      FUNCTION_BLOCK FB_Scheduler_F21
      VAR_INPUT
          currH : WORD;
          currM : WORD;
          currD : WORD;
      END_VAR
      VAR_IN_OUT
          FB_Bacnet : FB_BACnet_DAIKIN_MasterStation_III_No_5;
          FB_Bacnet_b : FB_BACnet_DAIKIN_MasterStation_III_No_6;
      END_VAR
      VAR
          i : INT;
          bUnitTriggered : BOOL := FALSE; // New flag to track execution
          prevMinute : WORD := 0;        // New variable to track the previous minute
      END_VAR
      VAR PERSISTENT
          //scheduler var
          bEnSchedF21_ : BOOL := FALSE;
          wSchedWDHourStartF21_ : WORD; 
          wSchedWDMinStartF21_ : WORD; 
          wSchedWEHourStartF21_ : WORD; 
          wSchedWEMinStartF21_ : WORD;
          wSchedWDHourEndF21_ : WORD;
          wSchedWDMinEndF21_ : WORD;
          wSchedWEHourEndF21_ : WORD;
          wSchedWEMinEndF21_ : WORD;
          //unit var
          bUnitF21_ : ARRAY [1..23] OF BOOL;
      END_VAR


        // Reset trigger flag at minute change or at the exact scheduled time
        IF currM <> prevMinute OR 
           (currH = wSchedWDHourStartF21_ AND currM = wSchedWDMinStartF21_) OR 
           (currH = wSchedWDHourEndF21_ AND currM = wSchedWDMinEndF21_) THEN
            bUnitTriggered := FALSE;
            prevMinute := currM;
        END_IF

        // Unit Schedule Enable
        IF bEnSchedF21_ THEN
            // Weekday schedule
            IF currD >= 1 AND currD <= 5 THEN
                IF (wSchedWDHourStartF21_ <> wSchedWDHourEndF21_ OR wSchedWDMinStartF21_ <> wSchedWDMinEndF21_) THEN
                    // Schedule Unit ON
                    IF wSchedWDHourStartF21_ = currH AND wSchedWDMinStartF21_ = currM AND NOT bUnitTriggered THEN
                        bUnitTriggered := TRUE;
                        FOR i := 1 TO 23 DO
                            // Send command unit ON
                            IF bUnitF21_[i] THEN 
                                CASE i OF
                                    1: 
                                        
                                        FB_Bacnet.StartStopCommand_192.bEnWrite := TRUE;
                                        FB_Bacnet.StartStopCommand_192.bVal := TRUE;
                                    2: 
                                        
                                        FB_Bacnet.StartStopCommand_193.bEnWrite := TRUE;
                                        FB_Bacnet.StartStopCommand_193.bVal := TRUE;
                                    3: 
                                        
                                        FB_Bacnet.StartStopCommand_194.bEnWrite := TRUE;
                                        FB_Bacnet.StartStopCommand_194.bVal := TRUE;
                                    4: 
                                        
                                        FB_Bacnet.StartStopCommand_195.bEnWrite := TRUE;
                                        FB_Bacnet.StartStopCommand_195.bVal := TRUE;
                                    5: 
                                        
                                        FB_Bacnet.StartStopCommand_196.bEnWrite := TRUE;
                                        FB_Bacnet.StartStopCommand_196.bVal := TRUE;
                                    6: 
                                        
                                        FB_Bacnet.StartStopCommand_197.bEnWrite := TRUE;
                                        FB_Bacnet.StartStopCommand_197.bVal := TRUE;
                                    7: 
                                        
                                        FB_Bacnet.StartStopCommand_198.bEnWrite := TRUE;
                                        FB_Bacnet.StartStopCommand_198.bVal := TRUE;
                                    8: 
                                        
                                        FB_Bacnet.StartStopCommand_199.bEnWrite := TRUE;
                                        FB_Bacnet.StartStopCommand_199.bVal := TRUE;
                                    9: 
                                        
                                        FB_Bacnet.StartStopCommand_200.bEnWrite := TRUE;
                                        FB_Bacnet.StartStopCommand_200.bVal := TRUE;
                                    10: 
                                        
                                        FB_Bacnet.StartStopCommand_201.bEnWrite := TRUE;
                                        FB_Bacnet.StartStopCommand_201.bVal := TRUE;
                                    11: 
                                        
                                        FB_Bacnet.StartStopCommand_202.bEnWrite := TRUE;
                                        FB_Bacnet.StartStopCommand_202.bVal := TRUE;
                                    12: 
                                        
                                        FB_Bacnet.StartStopCommand_203.bEnWrite := TRUE;
                                        FB_Bacnet.StartStopCommand_203.bVal := TRUE;
                                    13: 
                                        
                                        FB_Bacnet.StartStopCommand_204.bEnWrite := TRUE;
                                        FB_Bacnet.StartStopCommand_204.bVal := TRUE;
                                    14: 
                                        
                                        FB_Bacnet.StartStopCommand_205.bEnWrite := TRUE;
                                        FB_Bacnet.StartStopCommand_205.bVal := TRUE;
                                    15: 
                                        
                                        FB_Bacnet.StartStopCommand_206.bEnWrite := TRUE;
                                        FB_Bacnet.StartStopCommand_206.bVal := TRUE;
                                    16: 
                                        
                                        FB_Bacnet.StartStopCommand_207.bEnWrite := TRUE;
                                        FB_Bacnet.StartStopCommand_207.bVal := TRUE;
                                    17: 
                                        
                                        FB_Bacnet.StartStopCommand_208.bEnWrite := TRUE;
                                        FB_Bacnet.StartStopCommand_208.bVal := TRUE;
                                    18: 
                                        
                                        FB_Bacnet.StartStopCommand_209.bEnWrite := TRUE;
                                        FB_Bacnet.StartStopCommand_209.bVal := TRUE;
                                    19: 
                                        
                                        FB_Bacnet.StartStopCommand_210.bEnWrite := TRUE;
                                        FB_Bacnet.StartStopCommand_210.bVal := TRUE;
                                    20: 
                                        
                                        FB_Bacnet.StartStopCommand_211.bEnWrite := TRUE;
                                        FB_Bacnet.StartStopCommand_211.bVal := TRUE;
                                    21: 
                                        
                                        FB_Bacnet.StartStopCommand_240.bEnWrite := TRUE;
                                        FB_Bacnet.StartStopCommand_240.bVal := TRUE;
                                    22: 
                                        
                                        FB_Bacnet_b.StartStopCommand_049.bEnWrite := TRUE;
                                        FB_Bacnet_b.StartStopCommand_049.bVal := TRUE;
                                    23: 
                                        
                                        FB_Bacnet_b.StartStopCommand_034.bEnWrite := TRUE;
                                        FB_Bacnet_b.StartStopCommand_034.bVal := TRUE;
                                END_CASE
                            END_IF
                        END_FOR
                    END_IF
                    // Schedule Unit OFF
                    IF wSchedWDHourEndF21_ = currH AND wSchedWDMinEndF21_ = currM AND NOT bUnitTriggered THEN
                        bUnitTriggered := TRUE;
                        FOR i := 1 TO 23 DO
                            // Send command unit OFF
                            IF bUnitF21_[i] THEN 
                                CASE i OF
                                    1: 
                                        
                                        FB_Bacnet.StartStopCommand_192.bEnWrite := TRUE;
                                        FB_Bacnet.StartStopCommand_192.bVal := FALSE;
                                    2: 
                                        
                                        FB_Bacnet.StartStopCommand_193.bEnWrite := TRUE;
                                        FB_Bacnet.StartStopCommand_193.bVal := FALSE;
                                    3: 
                                        
                                        FB_Bacnet.StartStopCommand_194.bEnWrite := TRUE;
                                        FB_Bacnet.StartStopCommand_194.bVal := FALSE;
                                    4: 
                                        
                                        FB_Bacnet.StartStopCommand_195.bEnWrite := TRUE;
                                        FB_Bacnet.StartStopCommand_195.bVal := FALSE;
                                    5: 
                                        
                                        FB_Bacnet.StartStopCommand_196.bEnWrite := TRUE;
                                        FB_Bacnet.StartStopCommand_196.bVal := FALSE;
                                    6: 
                                        
                                        FB_Bacnet.StartStopCommand_197.bEnWrite := TRUE;
                                        FB_Bacnet.StartStopCommand_197.bVal := FALSE;
                                    7: 
                                        
                                        FB_Bacnet.StartStopCommand_198.bEnWrite := TRUE;
                                        FB_Bacnet.StartStopCommand_198.bVal := FALSE;
                                    8: 
                                        
                                        FB_Bacnet.StartStopCommand_199.bEnWrite := TRUE;
                                        FB_Bacnet.StartStopCommand_199.bVal := FALSE;
                                    9: 
                                        
                                        FB_Bacnet.StartStopCommand_200.bEnWrite := TRUE;
                                        FB_Bacnet.StartStopCommand_200.bVal := FALSE;
                                    10: 
                                        
                                        FB_Bacnet.StartStopCommand_201.bEnWrite := TRUE;
                                        FB_Bacnet.StartStopCommand_201.bVal := FALSE;
                                    11: 
                                        
                                        FB_Bacnet.StartStopCommand_202.bEnWrite := TRUE;
                                        FB_Bacnet.StartStopCommand_202.bVal := FALSE;
                                    12: 
                                        
                                        FB_Bacnet.StartStopCommand_203.bEnWrite := TRUE;
                                        FB_Bacnet.StartStopCommand_203.bVal := FALSE;
                                    13: 
                                        
                                        FB_Bacnet.StartStopCommand_204.bEnWrite := TRUE;
                                        FB_Bacnet.StartStopCommand_204.bVal := FALSE;
                                    14: 
                                        
                                        FB_Bacnet.StartStopCommand_205.bEnWrite := TRUE;
                                        FB_Bacnet.StartStopCommand_205.bVal := FALSE;
                                    15: 
                                        
                                        FB_Bacnet.StartStopCommand_206.bEnWrite := TRUE;
                                        FB_Bacnet.StartStopCommand_206.bVal := FALSE;
                                    16: 
                                        
                                        FB_Bacnet.StartStopCommand_207.bEnWrite := TRUE;
                                        FB_Bacnet.StartStopCommand_207.bVal := FALSE;
                                    17: 
                                        
                                        FB_Bacnet.StartStopCommand_208.bEnWrite := TRUE;
                                        FB_Bacnet.StartStopCommand_208.bVal := FALSE;
                                    18: 
                                        
                                        FB_Bacnet.StartStopCommand_209.bEnWrite := TRUE;
                                        FB_Bacnet.StartStopCommand_209.bVal := FALSE;
                                    19: 
                                        
                                        FB_Bacnet.StartStopCommand_210.bEnWrite := TRUE;
                                        FB_Bacnet.StartStopCommand_210.bVal := FALSE;
                                    20: 
                                        
                                        FB_Bacnet.StartStopCommand_211.bEnWrite := TRUE;
                                        FB_Bacnet.StartStopCommand_211.bVal := FALSE;
                                    21: 
                                        
                                        FB_Bacnet.StartStopCommand_240.bEnWrite := TRUE;
                                        FB_Bacnet.StartStopCommand_240.bVal := FALSE;
                                    22: 
                                        
                                        FB_Bacnet_b.StartStopCommand_049.bEnWrite := TRUE;
                                        FB_Bacnet_b.StartStopCommand_049.bVal := FALSE;
                                    23: 
                                        
                                        FB_Bacnet_b.StartStopCommand_034.bEnWrite := TRUE;
                                        FB_Bacnet_b.StartStopCommand_034.bVal := FALSE;
                                END_CASE
                            END_IF
                        END_FOR
                    END_IF
                END_IF
            END_IF

            // Weekend schedule
            IF currD = 0 OR currD = 6 THEN
                IF (wSchedWEHourStartF21_ <> wSchedWEHourEndF21_ OR wSchedWEMinStartF21_ <> wSchedWEMinEndF21_) THEN
                    // Schedule Unit ON
                    IF wSchedWEHourStartF21_ = currH AND wSchedWEMinStartF21_ = currM AND NOT bUnitTriggered THEN
                        bUnitTriggered := TRUE;
                        FOR i := 1 TO 23 DO
                            // Send command unit ON
                            IF bUnitF21_[i] THEN 
                                CASE i OF
                                    1: 
                                        
                                        FB_Bacnet.StartStopCommand_192.bEnWrite := TRUE;
                                        FB_Bacnet.StartStopCommand_192.bVal := TRUE;
                                    2: 
                                        
                                        FB_Bacnet.StartStopCommand_193.bEnWrite := TRUE;
                                        FB_Bacnet.StartStopCommand_193.bVal := TRUE;
                                    3: 
                                        
                                        FB_Bacnet.StartStopCommand_194.bEnWrite := TRUE;
                                        FB_Bacnet.StartStopCommand_194.bVal := TRUE;
                                    4: 
                                        
                                        FB_Bacnet.StartStopCommand_195.bEnWrite := TRUE;
                                        FB_Bacnet.StartStopCommand_195.bVal := TRUE;
                                    5: 
                                        
                                        FB_Bacnet.StartStopCommand_196.bEnWrite := TRUE;
                                        FB_Bacnet.StartStopCommand_196.bVal := TRUE;
                                    6: 
                                        
                                        FB_Bacnet.StartStopCommand_197.bEnWrite := TRUE;
                                        FB_Bacnet.StartStopCommand_197.bVal := TRUE;
                                    7: 
                                        
                                        FB_Bacnet.StartStopCommand_198.bEnWrite := TRUE;
                                        FB_Bacnet.StartStopCommand_198.bVal := TRUE;
                                    8: 
                                        
                                        FB_Bacnet.StartStopCommand_199.bEnWrite := TRUE;
                                        FB_Bacnet.StartStopCommand_199.bVal := TRUE;
                                    9: 
                                        
                                        FB_Bacnet.StartStopCommand_200.bEnWrite := TRUE;
                                        FB_Bacnet.StartStopCommand_200.bVal := TRUE;
                                    10: 
                                        
                                        FB_Bacnet.StartStopCommand_201.bEnWrite := TRUE;
                                        FB_Bacnet.StartStopCommand_201.bVal := TRUE;
                                    11: 
                                        
                                        FB_Bacnet.StartStopCommand_202.bEnWrite := TRUE;
                                        FB_Bacnet.StartStopCommand_202.bVal := TRUE;
                                    12: 
                                        
                                        FB_Bacnet.StartStopCommand_203.bEnWrite := TRUE;
                                        FB_Bacnet.StartStopCommand_203.bVal := TRUE;
                                    13: 
                                        
                                        FB_Bacnet.StartStopCommand_204.bEnWrite := TRUE;
                                        FB_Bacnet.StartStopCommand_204.bVal := TRUE;
                                    14: 
                                        
                                        FB_Bacnet.StartStopCommand_205.bEnWrite := TRUE;
                                        FB_Bacnet.StartStopCommand_205.bVal := TRUE;
                                    15: 
                                        
                                        FB_Bacnet.StartStopCommand_206.bEnWrite := TRUE;
                                        FB_Bacnet.StartStopCommand_206.bVal := TRUE;
                                    16: 
                                        
                                        FB_Bacnet.StartStopCommand_207.bEnWrite := TRUE;
                                        FB_Bacnet.StartStopCommand_207.bVal := TRUE;
                                    17: 
                                        
                                        FB_Bacnet.StartStopCommand_208.bEnWrite := TRUE;
                                        FB_Bacnet.StartStopCommand_208.bVal := TRUE;
                                    18: 
                                        
                                        FB_Bacnet.StartStopCommand_209.bEnWrite := TRUE;
                                        FB_Bacnet.StartStopCommand_209.bVal := TRUE;
                                    19: 
                                        
                                        FB_Bacnet.StartStopCommand_210.bEnWrite := TRUE;
                                        FB_Bacnet.StartStopCommand_210.bVal := TRUE;
                                    20: 
                                        
                                        FB_Bacnet.StartStopCommand_211.bEnWrite := TRUE;
                                        FB_Bacnet.StartStopCommand_211.bVal := TRUE;
                                    21: 
                                        
                                        FB_Bacnet.StartStopCommand_240.bEnWrite := TRUE;
                                        FB_Bacnet.StartStopCommand_240.bVal := TRUE;
                                    22: 
                                        
                                        FB_Bacnet_b.StartStopCommand_049.bEnWrite := TRUE;
                                        FB_Bacnet_b.StartStopCommand_049.bVal := TRUE;
                                    23: 
                                        
                                        FB_Bacnet_b.StartStopCommand_034.bEnWrite := TRUE;
                                        FB_Bacnet_b.StartStopCommand_034.bVal := TRUE;
                                END_CASE
                            END_IF
                        END_FOR
                    END_IF
                    // Schedule Unit OFF
                    IF wSchedWEHourEndF21_ = currH AND wSchedWEMinEndF21_ = currM AND NOT bUnitTriggered THEN
                        bUnitTriggered := TRUE;
                        FOR i := 1 TO 23 DO
                            // Send command unit OFF
                            IF bUnitF21_[i] THEN 
                                CASE i OF
                                    1: 
                                        
                                        FB_Bacnet.StartStopCommand_192.bEnWrite := TRUE;
                                        FB_Bacnet.StartStopCommand_192.bVal := FALSE;
                                    2: 
                                        
                                        FB_Bacnet.StartStopCommand_193.bEnWrite := TRUE;
                                        FB_Bacnet.StartStopCommand_193.bVal := FALSE;
                                    3: 
                                        
                                        FB_Bacnet.StartStopCommand_194.bEnWrite := TRUE;
                                        FB_Bacnet.StartStopCommand_194.bVal := FALSE;
                                    4: 
                                        
                                        FB_Bacnet.StartStopCommand_195.bEnWrite := TRUE;
                                        FB_Bacnet.StartStopCommand_195.bVal := FALSE;
                                    5: 
                                        
                                        FB_Bacnet.StartStopCommand_196.bEnWrite := TRUE;
                                        FB_Bacnet.StartStopCommand_196.bVal := FALSE;
                                    6: 
                                        
                                        FB_Bacnet.StartStopCommand_197.bEnWrite := TRUE;
                                        FB_Bacnet.StartStopCommand_197.bVal := FALSE;
                                    7: 
                                        
                                        FB_Bacnet.StartStopCommand_198.bEnWrite := TRUE;
                                        FB_Bacnet.StartStopCommand_198.bVal := FALSE;
                                    8: 
                                        
                                        FB_Bacnet.StartStopCommand_199.bEnWrite := TRUE;
                                        FB_Bacnet.StartStopCommand_199.bVal := FALSE;
                                    9: 
                                        
                                        FB_Bacnet.StartStopCommand_200.bEnWrite := TRUE;
                                        FB_Bacnet.StartStopCommand_200.bVal := FALSE;
                                    10: 
                                        
                                        FB_Bacnet.StartStopCommand_201.bEnWrite := TRUE;
                                        FB_Bacnet.StartStopCommand_201.bVal := FALSE;
                                    11: 
                                        
                                        FB_Bacnet.StartStopCommand_202.bEnWrite := TRUE;
                                        FB_Bacnet.StartStopCommand_202.bVal := FALSE;
                                    12: 
                                        
                                        FB_Bacnet.StartStopCommand_203.bEnWrite := TRUE;
                                        FB_Bacnet.StartStopCommand_203.bVal := FALSE;
                                    13: 
                                        
                                        FB_Bacnet.StartStopCommand_204.bEnWrite := TRUE;
                                        FB_Bacnet.StartStopCommand_204.bVal := FALSE;
                                    14: 
                                        
                                        FB_Bacnet.StartStopCommand_205.bEnWrite := TRUE;
                                        FB_Bacnet.StartStopCommand_205.bVal := FALSE;
                                    15: 
                                        
                                        FB_Bacnet.StartStopCommand_206.bEnWrite := TRUE;
                                        FB_Bacnet.StartStopCommand_206.bVal := FALSE;
                                    16: 
                                        
                                        FB_Bacnet.StartStopCommand_207.bEnWrite := TRUE;
                                        FB_Bacnet.StartStopCommand_207.bVal := FALSE;
                                    17: 
                                        
                                        FB_Bacnet.StartStopCommand_208.bEnWrite := TRUE;
                                        FB_Bacnet.StartStopCommand_208.bVal := FALSE;
                                    18: 
                                        
                                        FB_Bacnet.StartStopCommand_209.bEnWrite := TRUE;
                                        FB_Bacnet.StartStopCommand_209.bVal := FALSE;
                                    19: 
                                        
                                        FB_Bacnet.StartStopCommand_210.bEnWrite := TRUE;
                                        FB_Bacnet.StartStopCommand_210.bVal := FALSE;
                                    20: 
                                        
                                        FB_Bacnet.StartStopCommand_211.bEnWrite := TRUE;
                                        FB_Bacnet.StartStopCommand_211.bVal := FALSE;
                                    21: 
                                        
                                        FB_Bacnet.StartStopCommand_240.bEnWrite := TRUE;
                                        FB_Bacnet.StartStopCommand_240.bVal := FALSE;
                                    22: 
                                        
                                        FB_Bacnet_b.StartStopCommand_049.bEnWrite := TRUE;
                                        FB_Bacnet_b.StartStopCommand_049.bVal := FALSE;
                                    23: 
                                        
                                        FB_Bacnet_b.StartStopCommand_034.bEnWrite := TRUE;
                                        FB_Bacnet_b.StartStopCommand_034.bVal := FALSE;
                                END_CASE
                            END_IF
                        END_FOR
                    END_IF
                END_IF
            END_IF
        END_IF

END_FUNCTION_BLOCK

// ---- POUs/FB_Scheduler/FB_Scheduler_F22.TcPOU

      FUNCTION_BLOCK FB_Scheduler_F22
      VAR_INPUT
          currH : WORD;
          currM : WORD;
          currD : WORD;
      END_VAR
      VAR_IN_OUT
          FB_Bacnet : FB_BACnet_DAIKIN_MasterStation_III_No_6;
      END_VAR
      VAR
          i : INT;
          bUnitTriggered : BOOL := FALSE; // New flag to track execution
          prevMinute : WORD := 0;        // New variable to track the previous minute
      END_VAR
      VAR PERSISTENT
          //scheduler var
          bEnSchedF22_ : BOOL := FALSE;
          wSchedWDHourStartF22_ : WORD; 
          wSchedWDMinStartF22_ : WORD; 
          wSchedWEHourStartF22_ : WORD; 
          wSchedWEMinStartF22_ : WORD;
          wSchedWDHourEndF22_ : WORD;
          wSchedWDMinEndF22_ : WORD;
          wSchedWEHourEndF22_ : WORD;
          wSchedWEMinEndF22_ : WORD;
          //unit var
          bUnitF22_ : ARRAY [1..21] OF BOOL;
      END_VAR


        // Reset trigger flag at minute change or at the exact scheduled time
        IF currM <> prevMinute OR 
           (currH = wSchedWDHourStartF22_ AND currM = wSchedWDMinStartF22_) OR 
           (currH = wSchedWDHourEndF22_ AND currM = wSchedWDMinEndF22_) THEN
            bUnitTriggered := FALSE;
            prevMinute := currM;
        END_IF

        // Unit Schedule Enable
        IF bEnSchedF22_ THEN
            // Weekday schedule
            IF currD >= 1 AND currD <= 5 THEN
                IF (wSchedWDHourStartF22_ <> wSchedWDHourEndF22_ OR wSchedWDMinStartF22_ <> wSchedWDMinEndF22_) THEN
                    // Schedule Unit ON
                    IF wSchedWDHourStartF22_ = currH AND wSchedWDMinStartF22_ = currM AND NOT bUnitTriggered THEN
                        bUnitTriggered := TRUE;
                        FOR i := 1 TO 21 DO
                            // Send command unit ON
                            IF bUnitF22_[i] THEN 
                                CASE i OF
                                    1: 
                                        
                                        FB_Bacnet.StartStopCommand_000.bEnWrite := TRUE;
                                        FB_Bacnet.StartStopCommand_000.bVal := TRUE;
                                    2: 
                                        
                                        FB_Bacnet.StartStopCommand_001.bEnWrite := TRUE;
                                        FB_Bacnet.StartStopCommand_001.bVal := TRUE;
                                    3: 
                                        
                                        FB_Bacnet.StartStopCommand_002.bEnWrite := TRUE;
                                        FB_Bacnet.StartStopCommand_002.bVal := TRUE;
                                    4: 
                                        
                                        FB_Bacnet.StartStopCommand_003.bEnWrite := TRUE;
                                        FB_Bacnet.StartStopCommand_003.bVal := TRUE;
                                    5: 
                                        
                                        FB_Bacnet.StartStopCommand_004.bEnWrite := TRUE;
                                        FB_Bacnet.StartStopCommand_004.bVal := TRUE;
                                    6: 
                                        
                                        FB_Bacnet.StartStopCommand_005.bEnWrite := TRUE;
                                        FB_Bacnet.StartStopCommand_005.bVal := TRUE;
                                    7: 
                                        
                                        FB_Bacnet.StartStopCommand_006.bEnWrite := TRUE;
                                        FB_Bacnet.StartStopCommand_006.bVal := TRUE;
                                    8: 
                                        
                                        FB_Bacnet.StartStopCommand_007.bEnWrite := TRUE;
                                        FB_Bacnet.StartStopCommand_007.bVal := TRUE;
                                    9: 
                                        
                                        FB_Bacnet.StartStopCommand_008.bEnWrite := TRUE;
                                        FB_Bacnet.StartStopCommand_008.bVal := TRUE;
                                    10: 
                                        
                                        FB_Bacnet.StartStopCommand_009.bEnWrite := TRUE;
                                        FB_Bacnet.StartStopCommand_009.bVal := TRUE;
                                    11: 
                                        
                                        FB_Bacnet.StartStopCommand_010.bEnWrite := TRUE;
                                        FB_Bacnet.StartStopCommand_010.bVal := TRUE;
                                    12: 
                                        
                                        FB_Bacnet.StartStopCommand_011.bEnWrite := TRUE;
                                        FB_Bacnet.StartStopCommand_011.bVal := TRUE;
                                    13: 
                                        
                                        FB_Bacnet.StartStopCommand_012.bEnWrite := TRUE;
                                        FB_Bacnet.StartStopCommand_012.bVal := TRUE;
                                    14: 
                                        
                                        FB_Bacnet.StartStopCommand_013.bEnWrite := TRUE;
                                        FB_Bacnet.StartStopCommand_013.bVal := TRUE;
                                    15: 
                                        
                                        FB_Bacnet.StartStopCommand_014.bEnWrite := TRUE;
                                        FB_Bacnet.StartStopCommand_014.bVal := TRUE;
                                    16: 
                                        
                                        FB_Bacnet.StartStopCommand_015.bEnWrite := TRUE;
                                        FB_Bacnet.StartStopCommand_015.bVal := TRUE;
                                    17: 
                                        
                                        FB_Bacnet.StartStopCommand_016.bEnWrite := TRUE;
                                        FB_Bacnet.StartStopCommand_016.bVal := TRUE;
                                    18: 
                                        
                                        FB_Bacnet.StartStopCommand_017.bEnWrite := TRUE;
                                        FB_Bacnet.StartStopCommand_017.bVal := TRUE;
                                    19: 
                                        
                                        FB_Bacnet.StartStopCommand_018.bEnWrite := TRUE;
                                        FB_Bacnet.StartStopCommand_018.bVal := TRUE;
                                    20: 
                                        
                                        FB_Bacnet.StartStopCommand_019.bEnWrite := TRUE;
                                        FB_Bacnet.StartStopCommand_019.bVal := TRUE;
                                    21: 
                                        
                                        FB_Bacnet.StartStopCommand_035.bEnWrite := TRUE;
                                        FB_Bacnet.StartStopCommand_035.bVal := TRUE;
                                END_CASE
                            END_IF
                        END_FOR
                    END_IF
                    // Schedule Unit OFF
                    IF wSchedWDHourEndF22_ = currH AND wSchedWDMinEndF22_ = currM AND NOT bUnitTriggered THEN
                        bUnitTriggered := TRUE;
                        FOR i := 1 TO 21 DO
                            // Send command unit OFF
                            IF bUnitF22_[i] THEN 
                                CASE i OF
                                    1: 
                                        
                                        FB_Bacnet.StartStopCommand_000.bEnWrite := TRUE;
                                        FB_Bacnet.StartStopCommand_000.bVal := FALSE;
                                    2: 
                                        
                                        FB_Bacnet.StartStopCommand_001.bEnWrite := TRUE;
                                        FB_Bacnet.StartStopCommand_001.bVal := FALSE;
                                    3: 
                                        
                                        FB_Bacnet.StartStopCommand_002.bEnWrite := TRUE;
                                        FB_Bacnet.StartStopCommand_002.bVal := FALSE;
                                    4: 
                                        
                                        FB_Bacnet.StartStopCommand_003.bEnWrite := TRUE;
                                        FB_Bacnet.StartStopCommand_003.bVal := FALSE;
                                    5: 
                                        
                                        FB_Bacnet.StartStopCommand_004.bEnWrite := TRUE;
                                        FB_Bacnet.StartStopCommand_004.bVal := FALSE;
                                    6: 
                                        
                                        FB_Bacnet.StartStopCommand_005.bEnWrite := TRUE;
                                        FB_Bacnet.StartStopCommand_005.bVal := FALSE;
                                    7: 
                                        
                                        FB_Bacnet.StartStopCommand_006.bEnWrite := TRUE;
                                        FB_Bacnet.StartStopCommand_006.bVal := FALSE;
                                    8: 
                                        
                                        FB_Bacnet.StartStopCommand_007.bEnWrite := TRUE;
                                        FB_Bacnet.StartStopCommand_007.bVal := FALSE;
                                    9: 
                                        
                                        FB_Bacnet.StartStopCommand_008.bEnWrite := TRUE;
                                        FB_Bacnet.StartStopCommand_008.bVal := FALSE;
                                    10: 
                                        
                                        FB_Bacnet.StartStopCommand_009.bEnWrite := TRUE;
                                        FB_Bacnet.StartStopCommand_009.bVal := FALSE;
                                    11: 
                                        
                                        FB_Bacnet.StartStopCommand_010.bEnWrite := TRUE;
                                        FB_Bacnet.StartStopCommand_010.bVal := FALSE;
                                    12: 
                                        
                                        FB_Bacnet.StartStopCommand_011.bEnWrite := TRUE;
                                        FB_Bacnet.StartStopCommand_011.bVal := FALSE;
                                    13: 
                                        
                                        FB_Bacnet.StartStopCommand_012.bEnWrite := TRUE;
                                        FB_Bacnet.StartStopCommand_012.bVal := FALSE;
                                    14: 
                                        
                                        FB_Bacnet.StartStopCommand_013.bEnWrite := TRUE;
                                        FB_Bacnet.StartStopCommand_013.bVal := FALSE;
                                    15: 
                                        
                                        FB_Bacnet.StartStopCommand_014.bEnWrite := TRUE;
                                        FB_Bacnet.StartStopCommand_014.bVal := FALSE;
                                    16: 
                                        
                                        FB_Bacnet.StartStopCommand_015.bEnWrite := TRUE;
                                        FB_Bacnet.StartStopCommand_015.bVal := FALSE;
                                    17: 
                                        
                                        FB_Bacnet.StartStopCommand_016.bEnWrite := TRUE;
                                        FB_Bacnet.StartStopCommand_016.bVal := FALSE;
                                    18: 
                                        
                                        FB_Bacnet.StartStopCommand_017.bEnWrite := TRUE;
                                        FB_Bacnet.StartStopCommand_017.bVal := FALSE;
                                    19: 
                                        
                                        FB_Bacnet.StartStopCommand_018.bEnWrite := TRUE;
                                        FB_Bacnet.StartStopCommand_018.bVal := FALSE;
                                    20: 
                                        
                                        FB_Bacnet.StartStopCommand_019.bEnWrite := TRUE;
                                        FB_Bacnet.StartStopCommand_019.bVal := FALSE;
                                    21: 
                                        
                                        FB_Bacnet.StartStopCommand_035.bEnWrite := TRUE;
                                        FB_Bacnet.StartStopCommand_035.bVal := FALSE;
                                END_CASE
                            END_IF
                        END_FOR
                    END_IF
                END_IF
            END_IF

            // Weekend schedule
            IF currD = 0 OR currD = 6 THEN
                IF (wSchedWEHourStartF22_ <> wSchedWEHourEndF22_ OR wSchedWEMinStartF22_ <> wSchedWEMinEndF22_) THEN
                    // Schedule Unit ON
                    IF wSchedWEHourStartF22_ = currH AND wSchedWEMinStartF22_ = currM AND NOT bUnitTriggered THEN
                        bUnitTriggered := TRUE;
                        FOR i := 1 TO 21 DO
                            // Send command unit ON
                            IF bUnitF22_[i] THEN 
                                CASE i OF
                                    1: 
                                        
                                        FB_Bacnet.StartStopCommand_000.bEnWrite := TRUE;
                                        FB_Bacnet.StartStopCommand_000.bVal := TRUE;
                                    2: 
                                        
                                        FB_Bacnet.StartStopCommand_001.bEnWrite := TRUE;
                                        FB_Bacnet.StartStopCommand_001.bVal := TRUE;
                                    3: 
                                        
                                        FB_Bacnet.StartStopCommand_002.bEnWrite := TRUE;
                                        FB_Bacnet.StartStopCommand_002.bVal := TRUE;
                                    4: 
                                        
                                        FB_Bacnet.StartStopCommand_003.bEnWrite := TRUE;
                                        FB_Bacnet.StartStopCommand_003.bVal := TRUE;
                                    5: 
                                        
                                        FB_Bacnet.StartStopCommand_004.bEnWrite := TRUE;
                                        FB_Bacnet.StartStopCommand_004.bVal := TRUE;
                                    6: 
                                        
                                        FB_Bacnet.StartStopCommand_005.bEnWrite := TRUE;
                                        FB_Bacnet.StartStopCommand_005.bVal := TRUE;
                                    7: 
                                        
                                        FB_Bacnet.StartStopCommand_006.bEnWrite := TRUE;
                                        FB_Bacnet.StartStopCommand_006.bVal := TRUE;
                                    8: 
                                        
                                        FB_Bacnet.StartStopCommand_007.bEnWrite := TRUE;
                                        FB_Bacnet.StartStopCommand_007.bVal := TRUE;
                                    9: 
                                        
                                        FB_Bacnet.StartStopCommand_008.bEnWrite := TRUE;
                                        FB_Bacnet.StartStopCommand_008.bVal := TRUE;
                                    10: 
                                        
                                        FB_Bacnet.StartStopCommand_009.bEnWrite := TRUE;
                                        FB_Bacnet.StartStopCommand_009.bVal := TRUE;
                                    11: 
                                        
                                        FB_Bacnet.StartStopCommand_010.bEnWrite := TRUE;
                                        FB_Bacnet.StartStopCommand_010.bVal := TRUE;
                                    12: 
                                        
                                        FB_Bacnet.StartStopCommand_011.bEnWrite := TRUE;
                                        FB_Bacnet.StartStopCommand_011.bVal := TRUE;
                                    13: 
                                        
                                        FB_Bacnet.StartStopCommand_012.bEnWrite := TRUE;
                                        FB_Bacnet.StartStopCommand_012.bVal := TRUE;
                                    14: 
                                        
                                        FB_Bacnet.StartStopCommand_013.bEnWrite := TRUE;
                                        FB_Bacnet.StartStopCommand_013.bVal := TRUE;
                                    15: 
                                        
                                        FB_Bacnet.StartStopCommand_014.bEnWrite := TRUE;
                                        FB_Bacnet.StartStopCommand_014.bVal := TRUE;
                                    16: 
                                        
                                        FB_Bacnet.StartStopCommand_015.bEnWrite := TRUE;
                                        FB_Bacnet.StartStopCommand_015.bVal := TRUE;
                                    17: 
                                        
                                        FB_Bacnet.StartStopCommand_016.bEnWrite := TRUE;
                                        FB_Bacnet.StartStopCommand_016.bVal := TRUE;
                                    18: 
                                        
                                        FB_Bacnet.StartStopCommand_017.bEnWrite := TRUE;
                                        FB_Bacnet.StartStopCommand_017.bVal := TRUE;
                                    19: 
                                        
                                        FB_Bacnet.StartStopCommand_018.bEnWrite := TRUE;
                                        FB_Bacnet.StartStopCommand_018.bVal := TRUE;
                                    20: 
                                        
                                        FB_Bacnet.StartStopCommand_019.bEnWrite := TRUE;
                                        FB_Bacnet.StartStopCommand_019.bVal := TRUE;
                                    21: 
                                        
                                        FB_Bacnet.StartStopCommand_035.bEnWrite := TRUE;
                                        FB_Bacnet.StartStopCommand_035.bVal := TRUE;
                                END_CASE
                            END_IF
                        END_FOR        
                    END_IF
                    // Schedule Unit OFF
                    IF wSchedWEHourEndF22_ = currH AND wSchedWEMinEndF22_ = currM AND NOT bUnitTriggered THEN
                        bUnitTriggered := TRUE;
                        FOR i := 1 TO 21 DO
                            // Send command unit OFF
                            IF bUnitF22_[i] THEN 
                                CASE i OF
                                    1: 
                                        
                                        FB_Bacnet.StartStopCommand_000.bEnWrite := TRUE;
                                        FB_Bacnet.StartStopCommand_000.bVal := FALSE;
                                    2: 
                                        
                                        FB_Bacnet.StartStopCommand_001.bEnWrite := TRUE;
                                        FB_Bacnet.StartStopCommand_001.bVal := FALSE;
                                    3: 
                                        
                                        FB_Bacnet.StartStopCommand_002.bEnWrite := TRUE;
                                        FB_Bacnet.StartStopCommand_002.bVal := FALSE;
                                    4: 
                                        
                                        FB_Bacnet.StartStopCommand_003.bEnWrite := TRUE;
                                        FB_Bacnet.StartStopCommand_003.bVal := FALSE;
                                    5: 
                                        
                                        FB_Bacnet.StartStopCommand_004.bEnWrite := TRUE;
                                        FB_Bacnet.StartStopCommand_004.bVal := FALSE;
                                    6: 
                                        
                                        FB_Bacnet.StartStopCommand_005.bEnWrite := TRUE;
                                        FB_Bacnet.StartStopCommand_005.bVal := FALSE;
                                    7: 
                                        
                                        FB_Bacnet.StartStopCommand_006.bEnWrite := TRUE;
                                        FB_Bacnet.StartStopCommand_006.bVal := FALSE;
                                    8: 
                                        
                                        FB_Bacnet.StartStopCommand_007.bEnWrite := TRUE;
                                        FB_Bacnet.StartStopCommand_007.bVal := FALSE;
                                    9: 
                                        
                                        FB_Bacnet.StartStopCommand_008.bEnWrite := TRUE;
                                        FB_Bacnet.StartStopCommand_008.bVal := FALSE;
                                    10: 
                                        
                                        FB_Bacnet.StartStopCommand_009.bEnWrite := TRUE;
                                        FB_Bacnet.StartStopCommand_009.bVal := FALSE;
                                    11: 
                                        
                                        FB_Bacnet.StartStopCommand_010.bEnWrite := TRUE;
                                        FB_Bacnet.StartStopCommand_010.bVal := FALSE;
                                    12: 
                                        
                                        FB_Bacnet.StartStopCommand_011.bEnWrite := TRUE;
                                        FB_Bacnet.StartStopCommand_011.bVal := FALSE;
                                    13: 
                                        
                                        FB_Bacnet.StartStopCommand_012.bEnWrite := TRUE;
                                        FB_Bacnet.StartStopCommand_012.bVal := FALSE;
                                    14: 
                                        
                                        FB_Bacnet.StartStopCommand_013.bEnWrite := TRUE;
                                        FB_Bacnet.StartStopCommand_013.bVal := FALSE;
                                    15: 
                                        
                                        FB_Bacnet.StartStopCommand_014.bEnWrite := TRUE;
                                        FB_Bacnet.StartStopCommand_014.bVal := FALSE;
                                    16: 
                                        
                                        FB_Bacnet.StartStopCommand_015.bEnWrite := TRUE;
                                        FB_Bacnet.StartStopCommand_015.bVal := FALSE;
                                    17: 
                                        
                                        FB_Bacnet.StartStopCommand_016.bEnWrite := TRUE;
                                        FB_Bacnet.StartStopCommand_016.bVal := FALSE;
                                    18: 
                                        
                                        FB_Bacnet.StartStopCommand_017.bEnWrite := TRUE;
                                        FB_Bacnet.StartStopCommand_017.bVal := FALSE;
                                    19: 
                                        
                                        FB_Bacnet.StartStopCommand_018.bEnWrite := TRUE;
                                        FB_Bacnet.StartStopCommand_018.bVal := FALSE;
                                    20: 
                                        
                                        FB_Bacnet.StartStopCommand_019.bEnWrite := TRUE;
                                        FB_Bacnet.StartStopCommand_019.bVal := FALSE;
                                    21: 
                                        
                                        FB_Bacnet.StartStopCommand_035.bEnWrite := TRUE;
                                        FB_Bacnet.StartStopCommand_035.bVal := FALSE;
                                END_CASE
                            END_IF
                        END_FOR
                    END_IF
                END_IF
            END_IF
        END_IF

END_FUNCTION_BLOCK

// ---- POUs/FB_Scheduler/FB_Scheduler_F23.TcPOU

      FUNCTION_BLOCK FB_Scheduler_F23
      VAR_INPUT
          currH : WORD;
          currM : WORD;
          currD : WORD;
      END_VAR
      VAR_IN_OUT
          FB_Bacnet : FB_BACnet_DAIKIN_MasterStation_III_No_6;
      END_VAR
      VAR
          i : INT;
          bUnitTriggered : BOOL := FALSE; // New flag to track execution
          prevMinute : WORD := 0;        // New variable to track the previous minute
      END_VAR
      VAR PERSISTENT
          //scheduler var
          bEnSchedF23_ : BOOL := FALSE;
          wSchedWDHourStartF23_ : WORD; 
          wSchedWDMinStartF23_ : WORD; 
          wSchedWEHourStartF23_ : WORD; 
          wSchedWEMinStartF23_ : WORD;
          wSchedWDHourEndF23_ : WORD;
          wSchedWDMinEndF23_ : WORD;
          wSchedWEHourEndF23_ : WORD;
          wSchedWEMinEndF23_ : WORD;
          //unit var
          bUnitF23_ : ARRAY [1..21] OF BOOL;
      END_VAR


        // Reset trigger flag at minute change or at the exact scheduled time
        IF currM <> prevMinute OR 
           (currH = wSchedWDHourStartF23_ AND currM = wSchedWDMinStartF23_) OR 
           (currH = wSchedWDHourEndF23_ AND currM = wSchedWDMinEndF23_) THEN
            bUnitTriggered := FALSE;
            prevMinute := currM;
        END_IF

        // Unit Schedule Enable
        IF bEnSchedF23_ THEN
            // Weekday schedule
            IF currD >= 1 AND currD <= 5 THEN
                IF (wSchedWDHourStartF23_ <> wSchedWDHourEndF23_ OR wSchedWDMinStartF23_ <> wSchedWDMinEndF23_) THEN
                    // Schedule Unit ON
                    IF wSchedWDHourStartF23_ = currH AND wSchedWDMinStartF23_ = currM AND NOT bUnitTriggered THEN
                        bUnitTriggered := TRUE;
                        FOR i := 1 TO 21 DO
                            // Send command unit ON
                            IF bUnitF23_[i] THEN 
                                CASE i OF
                                    1: 
                                        
                                        FB_Bacnet.StartStopCommand_064.bEnWrite := TRUE;
                                        FB_Bacnet.StartStopCommand_064.bVal := TRUE;
                                    2: 
                                        
                                        FB_Bacnet.StartStopCommand_065.bEnWrite := TRUE;
                                        FB_Bacnet.StartStopCommand_065.bVal := TRUE;
                                    3: 
                                        
                                        FB_Bacnet.StartStopCommand_066.bEnWrite := TRUE;
                                        FB_Bacnet.StartStopCommand_066.bVal := TRUE;
                                    4: 
                                        
                                        FB_Bacnet.StartStopCommand_067.bEnWrite := TRUE;
                                        FB_Bacnet.StartStopCommand_067.bVal := TRUE;
                                    5: 
                                        
                                        FB_Bacnet.StartStopCommand_068.bEnWrite := TRUE;
                                        FB_Bacnet.StartStopCommand_068.bVal := TRUE;
                                    6: 
                                        
                                        FB_Bacnet.StartStopCommand_069.bEnWrite := TRUE;
                                        FB_Bacnet.StartStopCommand_069.bVal := TRUE;
                                    7: 
                                        
                                        FB_Bacnet.StartStopCommand_070.bEnWrite := TRUE;
                                        FB_Bacnet.StartStopCommand_070.bVal := TRUE;
                                    8: 
                                        
                                        FB_Bacnet.StartStopCommand_071.bEnWrite := TRUE;
                                        FB_Bacnet.StartStopCommand_071.bVal := TRUE;
                                    9: 
                                        
                                        FB_Bacnet.StartStopCommand_072.bEnWrite := TRUE;
                                        FB_Bacnet.StartStopCommand_072.bVal := TRUE;
                                    10: 
                                        
                                        FB_Bacnet.StartStopCommand_073.bEnWrite := TRUE;
                                        FB_Bacnet.StartStopCommand_073.bVal := TRUE;
                                    11: 
                                        
                                        FB_Bacnet.StartStopCommand_074.bEnWrite := TRUE;
                                        FB_Bacnet.StartStopCommand_074.bVal := TRUE;
                                    12: 
                                        
                                        FB_Bacnet.StartStopCommand_075.bEnWrite := TRUE;
                                        FB_Bacnet.StartStopCommand_075.bVal := TRUE;
                                    13: 
                                        
                                        FB_Bacnet.StartStopCommand_076.bEnWrite := TRUE;
                                        FB_Bacnet.StartStopCommand_076.bVal := TRUE;
                                    14: 
                                        
                                        FB_Bacnet.StartStopCommand_077.bEnWrite := TRUE;
                                        FB_Bacnet.StartStopCommand_077.bVal := TRUE;
                                    15: 
                                        
                                        FB_Bacnet.StartStopCommand_078.bEnWrite := TRUE;
                                        FB_Bacnet.StartStopCommand_078.bVal := TRUE;
                                    16: 
                                        
                                        FB_Bacnet.StartStopCommand_079.bEnWrite := TRUE;
                                        FB_Bacnet.StartStopCommand_079.bVal := TRUE;
                                    17: 
                                        
                                        FB_Bacnet.StartStopCommand_080.bEnWrite := TRUE;
                                        FB_Bacnet.StartStopCommand_080.bVal := TRUE;
                                    18: 
                                        
                                        FB_Bacnet.StartStopCommand_081.bEnWrite := TRUE;
                                        FB_Bacnet.StartStopCommand_081.bVal := TRUE;
                                    19: 
                                        
                                        FB_Bacnet.StartStopCommand_082.bEnWrite := TRUE;
                                        FB_Bacnet.StartStopCommand_082.bVal := TRUE;
                                    20: 
                                        
                                        FB_Bacnet.StartStopCommand_083.bEnWrite := TRUE;
                                        FB_Bacnet.StartStopCommand_083.bVal := TRUE;
                                    21: 
                                        
                                        FB_Bacnet.StartStopCommand_224.bEnWrite := TRUE;
                                        FB_Bacnet.StartStopCommand_224.bVal := TRUE;
                                END_CASE
                            END_IF
                        END_FOR
                    END_IF
                    // Schedule Unit OFF
                    IF wSchedWDHourEndF23_ = currH AND wSchedWDMinEndF23_ = currM AND NOT bUnitTriggered THEN
                        bUnitTriggered := TRUE;
                        FOR i := 1 TO 21 DO
                            // Send command unit OFF
                            IF bUnitF23_[i] THEN 
                                CASE i OF
                                    1: 
                                        
                                        FB_Bacnet.StartStopCommand_064.bEnWrite := TRUE;
                                        FB_Bacnet.StartStopCommand_064.bVal := FALSE;
                                    2: 
                                        
                                        FB_Bacnet.StartStopCommand_065.bEnWrite := TRUE;
                                        FB_Bacnet.StartStopCommand_065.bVal := FALSE;
                                    3: 
                                        
                                        FB_Bacnet.StartStopCommand_066.bEnWrite := TRUE;
                                        FB_Bacnet.StartStopCommand_066.bVal := FALSE;
                                    4: 
                                        
                                        FB_Bacnet.StartStopCommand_067.bEnWrite := TRUE;
                                        FB_Bacnet.StartStopCommand_067.bVal := FALSE;
                                    5: 
                                        
                                        FB_Bacnet.StartStopCommand_068.bEnWrite := TRUE;
                                        FB_Bacnet.StartStopCommand_068.bVal := FALSE;
                                    6: 
                                        
                                        FB_Bacnet.StartStopCommand_069.bEnWrite := TRUE;
                                        FB_Bacnet.StartStopCommand_069.bVal := FALSE;
                                    7: 
                                        
                                        FB_Bacnet.StartStopCommand_070.bEnWrite := TRUE;
                                        FB_Bacnet.StartStopCommand_070.bVal := FALSE;
                                    8: 
                                        
                                        FB_Bacnet.StartStopCommand_071.bEnWrite := TRUE;
                                        FB_Bacnet.StartStopCommand_071.bVal := FALSE;
                                    9: 
                                        
                                        FB_Bacnet.StartStopCommand_072.bEnWrite := TRUE;
                                        FB_Bacnet.StartStopCommand_072.bVal := FALSE;
                                    10: 
                                        
                                        FB_Bacnet.StartStopCommand_073.bEnWrite := TRUE;
                                        FB_Bacnet.StartStopCommand_073.bVal := FALSE;
                                    11: 
                                        
                                        FB_Bacnet.StartStopCommand_074.bEnWrite := TRUE;
                                        FB_Bacnet.StartStopCommand_074.bVal := FALSE;
                                    12: 
                                        
                                        FB_Bacnet.StartStopCommand_075.bEnWrite := TRUE;
                                        FB_Bacnet.StartStopCommand_075.bVal := FALSE;
                                    13: 
                                        
                                        FB_Bacnet.StartStopCommand_076.bEnWrite := TRUE;
                                        FB_Bacnet.StartStopCommand_076.bVal := FALSE;
                                    14: 
                                        
                                        FB_Bacnet.StartStopCommand_077.bEnWrite := TRUE;
                                        FB_Bacnet.StartStopCommand_077.bVal := FALSE;
                                    15: 
                                        
                                        FB_Bacnet.StartStopCommand_078.bEnWrite := TRUE;
                                        FB_Bacnet.StartStopCommand_078.bVal := FALSE;
                                    16: 
                                        
                                        FB_Bacnet.StartStopCommand_079.bEnWrite := TRUE;
                                        FB_Bacnet.StartStopCommand_079.bVal := FALSE;
                                    17: 
                                        
                                        FB_Bacnet.StartStopCommand_080.bEnWrite := TRUE;
                                        FB_Bacnet.StartStopCommand_080.bVal := FALSE;
                                    18: 
                                        
                                        FB_Bacnet.StartStopCommand_081.bEnWrite := TRUE;
                                        FB_Bacnet.StartStopCommand_081.bVal := FALSE;
                                    19: 
                                        
                                        FB_Bacnet.StartStopCommand_082.bEnWrite := TRUE;
                                        FB_Bacnet.StartStopCommand_082.bVal := FALSE;
                                    20: 
                                        
                                        FB_Bacnet.StartStopCommand_083.bEnWrite := TRUE;
                                        FB_Bacnet.StartStopCommand_083.bVal := FALSE;
                                    21: 
                                        
                                        FB_Bacnet.StartStopCommand_224.bEnWrite := TRUE;
                                        FB_Bacnet.StartStopCommand_224.bVal := FALSE;
                                END_CASE
                            END_IF
                        END_FOR
                    END_IF
                END_IF
            END_IF

            // Weekend schedule
            IF currD = 0 OR currD = 6 THEN
                IF (wSchedWEHourStartF23_ <> wSchedWEHourEndF23_ OR wSchedWEMinStartF23_ <> wSchedWEMinEndF23_) THEN
                    // Schedule Unit ON
                    IF wSchedWEHourStartF23_ = currH AND wSchedWEMinStartF23_ = currM AND NOT bUnitTriggered THEN
                        bUnitTriggered := TRUE;
                        FOR i := 1 TO 21 DO
                            // Send command unit ON
                            IF bUnitF23_[i] THEN 
                                CASE i OF
                                    1: 
                                        
                                        FB_Bacnet.StartStopCommand_064.bEnWrite := TRUE;
                                        FB_Bacnet.StartStopCommand_064.bVal := TRUE;
                                    2: 
                                        
                                        FB_Bacnet.StartStopCommand_065.bEnWrite := TRUE;
                                        FB_Bacnet.StartStopCommand_065.bVal := TRUE;
                                    3: 
                                        
                                        FB_Bacnet.StartStopCommand_066.bEnWrite := TRUE;
                                        FB_Bacnet.StartStopCommand_066.bVal := TRUE;
                                    4: 
                                        
                                        FB_Bacnet.StartStopCommand_067.bEnWrite := TRUE;
                                        FB_Bacnet.StartStopCommand_067.bVal := TRUE;
                                    5: 
                                        
                                        FB_Bacnet.StartStopCommand_068.bEnWrite := TRUE;
                                        FB_Bacnet.StartStopCommand_068.bVal := TRUE;
                                    6: 
                                        
                                        FB_Bacnet.StartStopCommand_069.bEnWrite := TRUE;
                                        FB_Bacnet.StartStopCommand_069.bVal := TRUE;
                                    7: 
                                        
                                        FB_Bacnet.StartStopCommand_070.bEnWrite := TRUE;
                                        FB_Bacnet.StartStopCommand_070.bVal := TRUE;
                                    8: 
                                        
                                        FB_Bacnet.StartStopCommand_071.bEnWrite := TRUE;
                                        FB_Bacnet.StartStopCommand_071.bVal := TRUE;
                                    9: 
                                        
                                        FB_Bacnet.StartStopCommand_072.bEnWrite := TRUE;
                                        FB_Bacnet.StartStopCommand_072.bVal := TRUE;
                                    10: 
                                        
                                        FB_Bacnet.StartStopCommand_073.bEnWrite := TRUE;
                                        FB_Bacnet.StartStopCommand_073.bVal := TRUE;
                                    11: 
                                        
                                        FB_Bacnet.StartStopCommand_074.bEnWrite := TRUE;
                                        FB_Bacnet.StartStopCommand_074.bVal := TRUE;
                                    12: 
                                        
                                        FB_Bacnet.StartStopCommand_075.bEnWrite := TRUE;
                                        FB_Bacnet.StartStopCommand_075.bVal := TRUE;
                                    13: 
                                        
                                        FB_Bacnet.StartStopCommand_076.bEnWrite := TRUE;
                                        FB_Bacnet.StartStopCommand_076.bVal := TRUE;
                                    14: 
                                        
                                        FB_Bacnet.StartStopCommand_077.bEnWrite := TRUE;
                                        FB_Bacnet.StartStopCommand_077.bVal := TRUE;
                                    15: 
                                        
                                        FB_Bacnet.StartStopCommand_078.bEnWrite := TRUE;
                                        FB_Bacnet.StartStopCommand_078.bVal := TRUE;
                                    16: 
                                        
                                        FB_Bacnet.StartStopCommand_079.bEnWrite := TRUE;
                                        FB_Bacnet.StartStopCommand_079.bVal := TRUE;
                                    17: 
                                        
                                        FB_Bacnet.StartStopCommand_080.bEnWrite := TRUE;
                                        FB_Bacnet.StartStopCommand_080.bVal := TRUE;
                                    18: 
                                        
                                        FB_Bacnet.StartStopCommand_081.bEnWrite := TRUE;
                                        FB_Bacnet.StartStopCommand_081.bVal := TRUE;
                                    19: 
                                        
                                        FB_Bacnet.StartStopCommand_082.bEnWrite := TRUE;
                                        FB_Bacnet.StartStopCommand_082.bVal := TRUE;
                                    20: 
                                        
                                        FB_Bacnet.StartStopCommand_083.bEnWrite := TRUE;
                                        FB_Bacnet.StartStopCommand_083.bVal := TRUE;
                                    21: 
                                        
                                        FB_Bacnet.StartStopCommand_224.bEnWrite := TRUE;
                                        FB_Bacnet.StartStopCommand_224.bVal := TRUE;
                                END_CASE
                            END_IF
                        END_FOR
                    END_IF
                    // Schedule Unit OFF
                    IF wSchedWEHourEndF23_ = currH AND wSchedWEMinEndF23_ = currM AND NOT bUnitTriggered THEN
                        bUnitTriggered := TRUE;
                        FOR i := 1 TO 21 DO
                            // Send command unit OFF
                            IF bUnitF23_[i] THEN 
                                CASE i OF
                                    1: 
                                        
                                        FB_Bacnet.StartStopCommand_064.bEnWrite := TRUE;
                                        FB_Bacnet.StartStopCommand_064.bVal := FALSE;
                                    2: 
                                        
                                        FB_Bacnet.StartStopCommand_065.bEnWrite := TRUE;
                                        FB_Bacnet.StartStopCommand_065.bVal := FALSE;
                                    3: 
                                        
                                        FB_Bacnet.StartStopCommand_066.bEnWrite := TRUE;
                                        FB_Bacnet.StartStopCommand_066.bVal := FALSE;
                                    4: 
                                        
                                        FB_Bacnet.StartStopCommand_067.bEnWrite := TRUE;
                                        FB_Bacnet.StartStopCommand_067.bVal := FALSE;
                                    5: 
                                        
                                        FB_Bacnet.StartStopCommand_068.bEnWrite := TRUE;
                                        FB_Bacnet.StartStopCommand_068.bVal := FALSE;
                                    6: 
                                        
                                        FB_Bacnet.StartStopCommand_069.bEnWrite := TRUE;
                                        FB_Bacnet.StartStopCommand_069.bVal := FALSE;
                                    7: 
                                        
                                        FB_Bacnet.StartStopCommand_070.bEnWrite := TRUE;
                                        FB_Bacnet.StartStopCommand_070.bVal := FALSE;
                                    8: 
                                        
                                        FB_Bacnet.StartStopCommand_071.bEnWrite := TRUE;
                                        FB_Bacnet.StartStopCommand_071.bVal := FALSE;
                                    9: 
                                        
                                        FB_Bacnet.StartStopCommand_072.bEnWrite := TRUE;
                                        FB_Bacnet.StartStopCommand_072.bVal := FALSE;
                                    10: 
                                        
                                        FB_Bacnet.StartStopCommand_073.bEnWrite := TRUE;
                                        FB_Bacnet.StartStopCommand_073.bVal := FALSE;
                                    11: 
                                        
                                        FB_Bacnet.StartStopCommand_074.bEnWrite := TRUE;
                                        FB_Bacnet.StartStopCommand_074.bVal := FALSE;
                                    12: 
                                        
                                        FB_Bacnet.StartStopCommand_075.bEnWrite := TRUE;
                                        FB_Bacnet.StartStopCommand_075.bVal := FALSE;
                                    13: 
                                        
                                        FB_Bacnet.StartStopCommand_076.bEnWrite := TRUE;
                                        FB_Bacnet.StartStopCommand_076.bVal := FALSE;
                                    14: 
                                        
                                        FB_Bacnet.StartStopCommand_077.bEnWrite := TRUE;
                                        FB_Bacnet.StartStopCommand_077.bVal := FALSE;
                                    15: 
                                        
                                        FB_Bacnet.StartStopCommand_078.bEnWrite := TRUE;
                                        FB_Bacnet.StartStopCommand_078.bVal := FALSE;
                                    16: 
                                        
                                        FB_Bacnet.StartStopCommand_079.bEnWrite := TRUE;
                                        FB_Bacnet.StartStopCommand_079.bVal := FALSE;
                                    17: 
                                        
                                        FB_Bacnet.StartStopCommand_080.bEnWrite := TRUE;
                                        FB_Bacnet.StartStopCommand_080.bVal := FALSE;
                                    18: 
                                        
                                        FB_Bacnet.StartStopCommand_081.bEnWrite := TRUE;
                                        FB_Bacnet.StartStopCommand_081.bVal := FALSE;
                                    19: 
                                        
                                        FB_Bacnet.StartStopCommand_082.bEnWrite := TRUE;
                                        FB_Bacnet.StartStopCommand_082.bVal := FALSE;
                                    20: 
                                        
                                        FB_Bacnet.StartStopCommand_083.bEnWrite := TRUE;
                                        FB_Bacnet.StartStopCommand_083.bVal := FALSE;
                                    21: 
                                        
                                        FB_Bacnet.StartStopCommand_224.bEnWrite := TRUE;
                                        FB_Bacnet.StartStopCommand_224.bVal := FALSE;
                                END_CASE
                            END_IF
                        END_FOR
                    END_IF
                END_IF
            END_IF
        END_IF

END_FUNCTION_BLOCK

// ---- POUs/FB_Scheduler/FB_Scheduler_F25.TcPOU

      FUNCTION_BLOCK FB_Scheduler_F25
      VAR_INPUT
          currH : WORD;
          currM : WORD;
          currD : WORD;
      END_VAR
      VAR_IN_OUT
          FB_Bacnet : FB_BACnet_DAIKIN_MasterStation_III_No_6;
      END_VAR
      VAR
          i : INT;
          bUnitTriggered : BOOL := FALSE; // New flag to track execution
          prevMinute : WORD := 0;        // New variable to track the previous minute
      END_VAR
      VAR PERSISTENT
          //scheduler var
          bEnSchedF25_ : BOOL := FALSE;
          wSchedWDHourStartF25_ : WORD; 
          wSchedWDMinStartF25_ : WORD; 
          wSchedWEHourStartF25_ : WORD; 
          wSchedWEMinStartF25_ : WORD;
          wSchedWDHourEndF25_ : WORD;
          wSchedWDMinEndF25_ : WORD;
          wSchedWEHourEndF25_ : WORD;
          wSchedWEMinEndF25_ : WORD;
          //unit var
          bUnitF25_ : ARRAY [1..23] OF BOOL;
      END_VAR


        // Reset trigger flag at minute change or at the exact scheduled time
        IF currM <> prevMinute OR 
           (currH = wSchedWDHourStartF25_ AND currM = wSchedWDMinStartF25_) OR 
           (currH = wSchedWDHourEndF25_ AND currM = wSchedWDMinEndF25_) THEN
            bUnitTriggered := FALSE;
            prevMinute := currM;
        END_IF

        // Unit Schedule Enable
        IF bEnSchedF25_ THEN
            // Weekday schedule
            IF currD >= 1 AND currD <= 5 THEN
                IF (wSchedWDHourStartF25_ <> wSchedWDHourEndF25_ OR wSchedWDMinStartF25_ <> wSchedWDMinEndF25_) THEN
                    // Schedule Unit ON
                    IF wSchedWDHourStartF25_ = currH AND wSchedWDMinStartF25_ = currM AND NOT bUnitTriggered THEN
                        bUnitTriggered := TRUE;
                        FOR i := 1 TO 23 DO
                            // Send command unit ON
                            IF bUnitF25_[i] THEN 
                                CASE i OF
                                    1: 
                                        
                                        FB_Bacnet.StartStopCommand_128.bEnWrite := TRUE;
                                        FB_Bacnet.StartStopCommand_128.bVal := TRUE;
                                    2: 
                                        
                                        FB_Bacnet.StartStopCommand_129.bEnWrite := TRUE;
                                        FB_Bacnet.StartStopCommand_129.bVal := TRUE;
                                    3: 
                                        
                                        FB_Bacnet.StartStopCommand_130.bEnWrite := TRUE;
                                        FB_Bacnet.StartStopCommand_130.bVal := TRUE;
                                    4: 
                                        
                                        FB_Bacnet.StartStopCommand_131.bEnWrite := TRUE;
                                        FB_Bacnet.StartStopCommand_131.bVal := TRUE;
                                    5: 
                                        
                                        FB_Bacnet.StartStopCommand_132.bEnWrite := TRUE;
                                        FB_Bacnet.StartStopCommand_132.bVal := TRUE;
                                    6: 
                                        
                                        FB_Bacnet.StartStopCommand_133.bEnWrite := TRUE;
                                        FB_Bacnet.StartStopCommand_133.bVal := TRUE;
                                    7: 
                                        //
                                        //FB_Bacnet.StartStopCommand_134.bEnWrite := TRUE;
                                        //FB_Bacnet.StartStopCommand_134.bVal := TRUE;
                                    8: 
                                        //
                                        //FB_Bacnet.StartStopCommand_135.bEnWrite := TRUE;
                                        //FB_Bacnet.StartStopCommand_135.bVal := TRUE;
                                    9: 
                                        
                                        FB_Bacnet.StartStopCommand_136.bEnWrite := TRUE;
                                        FB_Bacnet.StartStopCommand_136.bVal := TRUE;
                                    10: 
                                        
                                        FB_Bacnet.StartStopCommand_137.bEnWrite := TRUE;
                                        FB_Bacnet.StartStopCommand_137.bVal := TRUE;
                                    11: 
                                        
                                        FB_Bacnet.StartStopCommand_138.bEnWrite := TRUE;
                                        FB_Bacnet.StartStopCommand_138.bVal := TRUE;
                                    12: 
                                        
                                        FB_Bacnet.StartStopCommand_139.bEnWrite := TRUE;
                                        FB_Bacnet.StartStopCommand_139.bVal := TRUE;
                                    13: 
                                        
                                        FB_Bacnet.StartStopCommand_140.bEnWrite := TRUE;
                                        FB_Bacnet.StartStopCommand_140.bVal := TRUE;
                                    14: 
                                        
                                        FB_Bacnet.StartStopCommand_141.bEnWrite := TRUE;
                                        FB_Bacnet.StartStopCommand_141.bVal := TRUE;
                                    15: 
                                        
                                        FB_Bacnet.StartStopCommand_142.bEnWrite := TRUE;
                                        FB_Bacnet.StartStopCommand_142.bVal := TRUE;
                                    16: 
                                        
                                        FB_Bacnet.StartStopCommand_143.bEnWrite := TRUE;
                                        FB_Bacnet.StartStopCommand_143.bVal := TRUE;
                                    17: 
                                        
                                        FB_Bacnet.StartStopCommand_144.bEnWrite := TRUE;
                                        FB_Bacnet.StartStopCommand_144.bVal := TRUE;
                                    18: 
                                        
                                        FB_Bacnet.StartStopCommand_145.bEnWrite := TRUE;
                                        FB_Bacnet.StartStopCommand_145.bVal := TRUE;
                                    19: 
                                        
                                        FB_Bacnet.StartStopCommand_146.bEnWrite := TRUE;
                                        FB_Bacnet.StartStopCommand_146.bVal := TRUE;
                                    20: 
                                        
                                        FB_Bacnet.StartStopCommand_147.bEnWrite := TRUE;
                                        FB_Bacnet.StartStopCommand_147.bVal := TRUE;
                                    21: 
                                        
                                        FB_Bacnet.StartStopCommand_176.bEnWrite := TRUE;
                                        FB_Bacnet.StartStopCommand_176.bVal := TRUE;
                                    22: 
                                        
                                        FB_Bacnet.StartStopCommand_241.bEnWrite := TRUE;
                                        FB_Bacnet.StartStopCommand_241.bVal := TRUE;
                                    23: 
                                        
                                        FB_Bacnet.StartStopCommand_225.bEnWrite := TRUE;
                                        FB_Bacnet.StartStopCommand_225.bVal := TRUE;
                                END_CASE
                            END_IF
                        END_FOR
                    END_IF
                    // Schedule Unit OFF
                    IF wSchedWDHourEndF25_ = currH AND wSchedWDMinEndF25_ = currM AND NOT bUnitTriggered THEN
                        bUnitTriggered := TRUE;
                        FOR i := 1 TO 23 DO
                            // Send command unit OFF
                            IF bUnitF25_[i] THEN 
                                CASE i OF
                                    1: 
                                        
                                        FB_Bacnet.StartStopCommand_128.bEnWrite := TRUE;
                                        FB_Bacnet.StartStopCommand_128.bVal := FALSE;
                                    2: 
                                        
                                        FB_Bacnet.StartStopCommand_129.bEnWrite := TRUE;
                                        FB_Bacnet.StartStopCommand_129.bVal := FALSE;
                                    3: 
                                        
                                        FB_Bacnet.StartStopCommand_130.bEnWrite := TRUE;
                                        FB_Bacnet.StartStopCommand_130.bVal := FALSE;
                                    4: 
                                        
                                        FB_Bacnet.StartStopCommand_131.bEnWrite := TRUE;
                                        FB_Bacnet.StartStopCommand_131.bVal := FALSE;
                                    5: 
                                        
                                        FB_Bacnet.StartStopCommand_132.bEnWrite := TRUE;
                                        FB_Bacnet.StartStopCommand_132.bVal := FALSE;
                                    6: 
                                        
                                        FB_Bacnet.StartStopCommand_133.bEnWrite := TRUE;
                                        FB_Bacnet.StartStopCommand_133.bVal := FALSE;
                                    7: 
                                        //
                                        //FB_Bacnet.StartStopCommand_134.bEnWrite := TRUE;
                                        //FB_Bacnet.StartStopCommand_134.bVal := FALSE;
                                    8: 
                                        //
                                        //FB_Bacnet.StartStopCommand_135.bEnWrite := TRUE;
                                        //FB_Bacnet.StartStopCommand_135.bVal := FALSE;
                                    9: 
                                        
                                        FB_Bacnet.StartStopCommand_136.bEnWrite := TRUE;
                                        FB_Bacnet.StartStopCommand_136.bVal := FALSE;
                                    10: 
                                        
                                        FB_Bacnet.StartStopCommand_137.bEnWrite := TRUE;
                                        FB_Bacnet.StartStopCommand_137.bVal := FALSE;
                                    11: 
                                        
                                        FB_Bacnet.StartStopCommand_138.bEnWrite := TRUE;
                                        FB_Bacnet.StartStopCommand_138.bVal := FALSE;
                                    12: 
                                        
                                        FB_Bacnet.StartStopCommand_139.bEnWrite := TRUE;
                                        FB_Bacnet.StartStopCommand_139.bVal := FALSE;
                                    13: 
                                        
                                        FB_Bacnet.StartStopCommand_140.bEnWrite := TRUE;
                                        FB_Bacnet.StartStopCommand_140.bVal := FALSE;
                                    14: 
                                        
                                        FB_Bacnet.StartStopCommand_141.bEnWrite := TRUE;
                                        FB_Bacnet.StartStopCommand_141.bVal := FALSE;
                                    15: 
                                        
                                        FB_Bacnet.StartStopCommand_142.bEnWrite := TRUE;
                                        FB_Bacnet.StartStopCommand_142.bVal := FALSE;
                                    16: 
                                        
                                        FB_Bacnet.StartStopCommand_143.bEnWrite := TRUE;
                                        FB_Bacnet.StartStopCommand_143.bVal := FALSE;
                                    17: 
                                        
                                        FB_Bacnet.StartStopCommand_144.bEnWrite := TRUE;
                                        FB_Bacnet.StartStopCommand_144.bVal := FALSE;
                                    18: 
                                        
                                        FB_Bacnet.StartStopCommand_145.bEnWrite := TRUE;
                                        FB_Bacnet.StartStopCommand_145.bVal := FALSE;
                                    19: 
                                        
                                        FB_Bacnet.StartStopCommand_146.bEnWrite := TRUE;
                                        FB_Bacnet.StartStopCommand_146.bVal := FALSE;
                                    20: 
                                        
                                        FB_Bacnet.StartStopCommand_147.bEnWrite := TRUE;
                                        FB_Bacnet.StartStopCommand_147.bVal := FALSE;
                                    21: 
                                        
                                        FB_Bacnet.StartStopCommand_176.bEnWrite := TRUE;
                                        FB_Bacnet.StartStopCommand_176.bVal := FALSE;
                                    22: 
                                        
                                        FB_Bacnet.StartStopCommand_241.bEnWrite := TRUE;
                                        FB_Bacnet.StartStopCommand_241.bVal := FALSE;
                                    23: 
                                        
                                        FB_Bacnet.StartStopCommand_225.bEnWrite := TRUE;
                                        FB_Bacnet.StartStopCommand_225.bVal := FALSE;
                                END_CASE
                            END_IF
                        END_FOR
                    END_IF
                END_IF
            END_IF

            // Weekend schedule
            IF currD = 0 OR currD = 6 THEN
                IF (wSchedWEHourStartF25_ <> wSchedWEHourEndF25_ OR wSchedWEMinStartF25_ <> wSchedWEMinEndF25_) THEN
                    // Schedule Unit ON
                    IF wSchedWEHourStartF25_ = currH AND wSchedWEMinStartF25_ = currM AND NOT bUnitTriggered THEN
                        bUnitTriggered := TRUE;
                        FOR i := 1 TO 23 DO
                            // Send command unit ON
                            IF bUnitF25_[i] THEN 
                                CASE i OF
                                    1: 
                                        
                                        FB_Bacnet.StartStopCommand_128.bEnWrite := TRUE;
                                        FB_Bacnet.StartStopCommand_128.bVal := TRUE;
                                    2: 
                                        
                                        FB_Bacnet.StartStopCommand_129.bEnWrite := TRUE;
                                        FB_Bacnet.StartStopCommand_129.bVal := TRUE;
                                    3: 
                                        
                                        FB_Bacnet.StartStopCommand_130.bEnWrite := TRUE;
                                        FB_Bacnet.StartStopCommand_130.bVal := TRUE;
                                    4: 
                                        
                                        FB_Bacnet.StartStopCommand_131.bEnWrite := TRUE;
                                        FB_Bacnet.StartStopCommand_131.bVal := TRUE;
                                    5: 
                                        
                                        FB_Bacnet.StartStopCommand_132.bEnWrite := TRUE;
                                        FB_Bacnet.StartStopCommand_132.bVal := TRUE;
                                    6: 
                                        
                                        FB_Bacnet.StartStopCommand_133.bEnWrite := TRUE;
                                        FB_Bacnet.StartStopCommand_133.bVal := TRUE;
                                    7: 
                                        //
                                        //FB_Bacnet.StartStopCommand_134.bEnWrite := TRUE;
                                        //FB_Bacnet.StartStopCommand_134.bVal := TRUE;
                                    8: 
                                        //
                                        //FB_Bacnet.StartStopCommand_135.bEnWrite := TRUE;
                                        //FB_Bacnet.StartStopCommand_135.bVal := TRUE;
                                    9: 
                                        
                                        FB_Bacnet.StartStopCommand_136.bEnWrite := TRUE;
                                        FB_Bacnet.StartStopCommand_136.bVal := TRUE;
                                    10: 
                                        
                                        FB_Bacnet.StartStopCommand_137.bEnWrite := TRUE;
                                        FB_Bacnet.StartStopCommand_137.bVal := TRUE;
                                    11: 
                                        
                                        FB_Bacnet.StartStopCommand_138.bEnWrite := TRUE;
                                        FB_Bacnet.StartStopCommand_138.bVal := TRUE;
                                    12: 
                                        
                                        FB_Bacnet.StartStopCommand_139.bEnWrite := TRUE;
                                        FB_Bacnet.StartStopCommand_139.bVal := TRUE;
                                    13: 
                                        
                                        FB_Bacnet.StartStopCommand_140.bEnWrite := TRUE;
                                        FB_Bacnet.StartStopCommand_140.bVal := TRUE;
                                    14: 
                                        
                                        FB_Bacnet.StartStopCommand_141.bEnWrite := TRUE;
                                        FB_Bacnet.StartStopCommand_141.bVal := TRUE;
                                    15: 
                                        
                                        FB_Bacnet.StartStopCommand_142.bEnWrite := TRUE;
                                        FB_Bacnet.StartStopCommand_142.bVal := TRUE;
                                    16: 
                                        
                                        FB_Bacnet.StartStopCommand_143.bEnWrite := TRUE;
                                        FB_Bacnet.StartStopCommand_143.bVal := TRUE;
                                    17: 
                                        
                                        FB_Bacnet.StartStopCommand_144.bEnWrite := TRUE;
                                        FB_Bacnet.StartStopCommand_144.bVal := TRUE;
                                    18: 
                                        
                                        FB_Bacnet.StartStopCommand_145.bEnWrite := TRUE;
                                        FB_Bacnet.StartStopCommand_145.bVal := TRUE;
                                    19: 
                                        
                                        FB_Bacnet.StartStopCommand_146.bEnWrite := TRUE;
                                        FB_Bacnet.StartStopCommand_146.bVal := TRUE;
                                    20: 
                                        
                                        FB_Bacnet.StartStopCommand_147.bEnWrite := TRUE;
                                        FB_Bacnet.StartStopCommand_147.bVal := TRUE;
                                    21: 
                                        
                                        FB_Bacnet.StartStopCommand_176.bEnWrite := TRUE;
                                        FB_Bacnet.StartStopCommand_176.bVal := TRUE;
                                    22: 
                                        
                                        FB_Bacnet.StartStopCommand_241.bEnWrite := TRUE;
                                        FB_Bacnet.StartStopCommand_241.bVal := TRUE;
                                    23: 
                                        
